INTERFACE I_AlarmManager

METHOD AcknowledgeAlarm : BOOL
VAR_INPUT
    nRecordId   : UDINT;
    sOperator   : STRING;
END_VAR
END_METHOD

METHOD ClearAlarm : BOOL
VAR_INPUT
    nRecordId : UDINT;
END_VAR
END_METHOD

METHOD GetActiveAlarmCount : INT
VAR_INPUT
END_VAR
END_METHOD

METHOD GetHighestAlarmLevel  : E_AlarmLevel
VAR_INPUT
END_VAR
END_METHOD

METHOD RaiseAlarm : BOOL
VAR_INPUT
    eLevel      : E_AlarmLevel;
    eZone       : E_ZoneId;
    nSensorId   : INT;
    rValue      : REAL;
    sDesc       : STRING;
END_VAR
END_METHOD

END_INTERFACE

(* stored: Version 1.1.0.1, ProductVersion 3.1.4024.16
   Itf I_AlarmManager: Id {e520ac3a-9e8e-4870-90ec-590559c3c100}
   Method AcknowledgeAlarm: Id {b3d76000-f9cb-4689-8f65-dba65dcf6edc}
   Method ClearAlarm: Id {01db593c-336c-402e-905f-9a9efdd00701}
   Method GetActiveAlarmCount: Id {009a0774-4251-420c-97b2-f33c6a3c2297}
   Method GetHighestAlarmLevel: Id {51eb67b8-8268-414c-abcb-ed3078b96579}
   Method RaiseAlarm: Id {fba0a1de-fc66-4689-8a49-2d6016a20876} *)
